FUNCTION_BLOCK MasterAxisControl
VAR
	
	_Axis			: AXIS_REF;
	
	_AnglePosition	: LREAL;
	_LengthOfShaft	: LREAL;
	_WidthOfShaft	: LREAL;
	_AxisSize		: LREAL;
	_xCoordRelative	: LREAL;
	_yCoordRelative	: LREAL;
	_LocalState		: BYTE;
	
	_Enable			: MC_Power;
	_Reset			: MC_Reset;
	_MovePosAbs		: MC_MoveAbsolute;
	_MovePosRel		: MC_MoveRelative;	
	_ReadStatus		: MC_ReadStatus;
	
END_VAR

PROPERTY AnglePosition : LREAL
GET
AnglePosition := _AnglePosition;
END_GET
SET
END_SET
END_PROPERTY

PROPERTY AxisSize : LREAL
GET
AxisSize := _AxisSize;
END_GET
SET
IF AxisSize < 0 THEN
	_AxisSize := 0;
ELSE
	_AxisSize := AxisSize;
END_IF
END_SET
END_PROPERTY

METHOD CyclicUpdate : BOOL
VAR_INPUT
END_VAR
_Enable(Axis := _Axis);
_Reset(Axis := _Axis);
_ReadStatus(Axis := _Axis);
_MovePosAbs(Axis := _Axis);
_MovePosRel(Axis := _Axis);

_AnglePosition := _Axis.NcToPlc.ModuloActPos;
END_METHOD

PROPERTY LengthOfShaft : LREAL
GET
LengthOfShaft := _LengthOfShaft;
END_GET
SET
IF LengthOfShaft < 0 THEN
	_LengthOfShaft := 0;
ELSE
	_LengthOfShaft := LengthOfShaft;
END_IF
END_SET
END_PROPERTY

METHOD MoveRelative : BOOL
VAR_INPUT
	Position	: LREAL;
	Velocity	: LREAL;
END_VAR
_MovePosRel(Axis := _Axis);
_MovePosRel.Distance := Position;
_MovePosRel.Velocity := Velocity;
_MovePosRel.Execute := TRUE;
IF _MovePosRel.Done THEN
	_MovePosRel.Execute := FALSE;
	MoveRelative := TRUE;
ELSIF _MovePosRel.Error THEN
	_MovePosRel.Execute := FALSE;
	MoveRelative := FALSE;
END_IF
END_METHOD

METHOD PowerOn : BOOL
VAR_INPUT
END_VAR
_Enable(Axis := _Axis);
_Enable.Enable := TRUE;
_Enable.Enable_Negative := TRUE;
_Enable.Enable_Positive := TRUE;
_Enable.Override := 100;
IF _Enable.Status THEN
	PowerOn := TRUE;
END_IF
END_METHOD

PROPERTY WidthOfShaft : LREAL
GET
WidthOfShaft := _WidthOfShaft;
END_GET
SET
IF WidthOfShaft < 0 THEN
	_WidthOfShaft := 0;
ELSE
	_WidthOfShaft := WidthOfShaft;
END_IF
END_SET
END_PROPERTY

PROPERTY XCoordRelative : LREAL
GET
XCoordRelative := _xCoordRelative;
END_GET
SET
_xCoordRelative := XCoordRelative;
END_SET
END_PROPERTY

PROPERTY YCoordRelative : LREAL
GET
YCoordRelative := _yCoordRelative;
END_GET
SET
_yCoordRelative := YCoordRelative;
END_SET
END_PROPERTY

END_FUNCTION_BLOCK

(* stored: Version 1.1.0.1, ProductVersion 3.1.4024.12
   POU MasterAxisControl: Id {06b8ec07-9351-4356-ad83-8beda64e605b}, SpecialFunc None
   Folder Methods: Id {55240223-bfe6-490d-877c-cceb4cbe873d}
   Folder Properties: Id {54f81e1e-9b88-4e2c-b721-85ee2157fbaf}
   Property AnglePosition: Id {a0efd3fa-6851-4f6d-bf5d-ab3919601722}
   Get Get: Id {e68dd914-bf5b-44d6-9d43-b2063d778c62}
   Set Set: Id {44a868f8-81ed-4547-bd40-1c7403f1f2b1}
   Property AxisSize: Id {3807e733-1314-49a8-98ee-94befc5ffa34}
   Get Get: Id {3dae204a-6b08-4d70-a24a-3b9e0ddada18}
   Set Set: Id {cb73dcfa-174b-4e7c-bf7b-975ed890d0ef}
   Method CyclicUpdate: Id {93cf9554-dd93-416c-9dfb-b77d81f9a9c7}
   Property LengthOfShaft: Id {0663e92e-7f49-4778-beae-8659eca01a4a}
   Get Get: Id {282f4c2d-1027-488d-94bd-9577e7af593e}
   Set Set: Id {3e643bf1-5234-4881-8fd3-0d7c97321420}
   Method MoveRelative: Id {ae23b31e-a597-4182-9778-44dab6fd606c}
   Method PowerOn: Id {4d1e9861-1256-4dab-b7e3-8aa6316c30d3}
   Property WidthOfShaft: Id {d2569453-f152-4749-bf99-e240475f1bac}
   Get Get: Id {4ed770ad-bf6e-4ad3-b2aa-cfb6834c3d50}
   Set Set: Id {f306815e-e89f-4876-a389-c901cd1024e0}
   Property XCoordRelative: Id {ac1e0834-41b4-4929-b6da-4d01ead02cbf}
   Get Get: Id {920133e8-80c4-4159-92fb-29f3d2eca0a4}
   Set Set: Id {40786f6d-2db5-4771-b814-271a0de52117}
   Property YCoordRelative: Id {2e91a015-1146-47df-af69-1be6e171815a}
   Get Get: Id {ca0037c2-f169-444d-b7c0-331d0e68b39b}
   Set Set: Id {800d9934-09e9-4796-b59f-0744426bbbe5} *)
